INTERFACE I_Session Extends I_Disposable

METHOD PUBLIC AddOrUpdateStorage
VAR_INPUT
	StorageId : T_MAXSTRING;
	Source : I_SessionData;
END_VAR
END_METHOD

METHOD PUBLIC DisposeAllDataFromStorage
VAR_INPUT
END_VAR
END_METHOD

METHOD PUBLIC DisposeDataFromStorage
VAR_INPUT
	StorageId : T_MAXSTRING;
END_VAR
END_METHOD

PROPERTY PUBLIC Id : T_MAXSTRING
GET
END_GET
END_PROPERTY

PROPERTY PUBLIC LastAccessedTimestamp : I_TimeStamp
GET
END_GET
END_PROPERTY

METHOD PUBLIC TryGetDataFromStorage : BOOL
VAR_INPUT
	StorageId : T_MAXSTRING;
	Destination : REFERENCE TO I_SessionData;
END_VAR
END_METHOD

END_INTERFACE

(* stored: Version 1.1.0.1, ProductVersion 3.1.4024.12
   Itf I_Session: Id {a9fc0945-06ac-49ad-b3d8-b714d5ead362}
   Method AddOrUpdateStorage: Id {ea7f5980-13f6-48ed-9b64-0ff46c27a765}
   Method DisposeAllDataFromStorage: Id {ce7e62fa-0352-429b-a636-e5b471c3dba0}
   Method DisposeDataFromStorage: Id {826a168b-6d7d-4b79-a327-319df8a3b56d}
   Property Id: Id {2ba75b52-1e1a-4e6e-859f-8c2dec2fe394}
   Get Get: Id {8188f276-7e24-4430-b432-da3febd3e3d8}
   Property LastAccessedTimestamp: Id {81103e14-8f0f-4123-ad4e-36a1a84dfaf7}
   Get Get: Id {57630843-6b99-4601-875e-70ec28963718}
   Method TryGetDataFromStorage: Id {2ae68a48-247d-4878-9606-cb764cdf35db} *)
